# EPICS StreamDevice protocol: GPD4303StestApp/Db/devGPD4303S.proto
ExtraInput = Ignore;
ReadTimeout = 100;
LockTimeout = 5000;
ReplyTimeout = 1000;

getIDN {
    out "*IDN?";
    in "%\$1[^\r\n]";
}

cmd {
    out "\$1";
}

setBoolean {
    out "\$1%{0|1}";
}

setDecimal {
    out "\$1%d";
}

getDecimal {
    out "\$1?";
    in "%d";
}

setFloat {
    out "\$1:%f";
}

getFloat {
    out "\$1?";
    in "%f";
}

setCurrentLimit {
    out "ISET1:%f";
    @init { out "ISET1?\r\n"; in "%f"; }
}
